RoboDK station: 250418.관통프로젝트준비파일.rdk

Station 250418.관통프로젝트준비파일 (saved by RoboDK 5.9.0). Poses are relative to the parent item; angles as X-Y-Z fixed-axis rotations.
  - Python program RESET (listed below)
  - Python program ADD_File (listed below)
  - notes Note 1: <!DOCTYPE HTML PUBLIC "-//W3C//DTD HTML 4.0//EN" "http://www.w3.org/TR/REC-html40/strict.dtd">
<html><head><meta name="qrichtext" content="1" /><style type="text/css">
p, li { white-space: pre-wrap; }
</style></head><body style=" font-family:'Gulim'; font-size:9pt; font-weight:400; font-style:normal;">
<p style=" margin-top:0px; margin-bottom:0px; margin-left:0px; margin-right:0px; -qt-block-indent:0; text-indent:0px;">관통프로젝트\모델링파일2을 모두 가져옵니다.</p>
<p style=" margin-top:0px; margin-bottom:0px; margin-left:0px; margin-right:0px; -qt-block-indent:0; text-indent:0px;">ADD_File을실행합니다.</p>
<p style=" margin-top:0px; margin-bottom:0px; margin-left:0px; margin-right:0px; -qt-block-indent:0; text-indent:0px;">RESET을 실행합니다.</p></body></html>

--- Python program RESET ---
from robodk import robolink    # RoboDK API
from robodk import robomath    # Robot toolbox
RDK = robolink.Robolink()
from robodk import *      # RoboDK API
from robolink import *    # Robot toolbox










Main_Frame=RDK.Item("Main_Frame",3)
Rack1_Frame=RDK.Item("Rack1 Base",3)
Rack2_Frame=RDK.Item("Rack2 Base",3)
Rack3_Frame=RDK.Item("Rack3 Base",3)
Rack4_Frame=RDK.Item("Rack4 Base",3)

Rack1=RDK.Item("Rack1",2)
Rack2=RDK.Item("Rack2",2)
Rack3=RDK.Item("Rack3",2)
Rack4=RDK.Item("Rack4",2)


Room=RDK.Item("Room",5)

def reset1(): #Room, Rack 위치 설정
      p1=[[     1.000000,     0.000000,     0.000000,     0.000000 ],
            [0.000000,     1.000000,     0.000000,     0.000000 ],
            [0.000000,     0.000000,     1.000000,     0.000000 ],
            [0.000000,     0.000000,     0.000000,     1.000000 ]]
      Room.setParent(Main_Frame)
      Room.setPose(Mat(p1))

      r1=[[     0.000000,     1.000000,     0.000000, -5000.000000 ],
      [-1.000000,     0.000000,     0.000000,  1000.000000 ],
            [0.000000,     0.000000,     1.000000,    50.000000 ],
            [0.000000,     0.000000,     0.000000,     1.000000 ]]


      Rack1_Frame.setPose(Mat(r1))
      Rack2_Frame.setPose(Mat(r1))
      Rack3_Frame.setPose(Mat(r1))
      Rack4_Frame.setPose(Mat(r1))

      Rack1_Frame.setParent(Main_Frame)
      Rack2_Frame.setParent(Main_Frame)
      Rack3_Frame.setParent(Main_Frame)
      Rack4_Frame.setParent(Main_Frame)


      Rack1.setParent(Rack1_Frame)
      Rack2.setParent(Rack2_Frame)
      Rack3.setParent(Rack3_Frame)
      Rack4.setParent(Rack4_Frame)



#####################################


CON1=RDK.Item("CON1",2)
CON1_Frame=RDK.Item("CON1 Base",3)
CON2=RDK.Item("CON2",2)
CON2_Frame=RDK.Item("CON2 Base",3)




def reset2(): #conveyor 위치 설정

      con_pos1=[[     1.000000,     0.000000,     0.000000,   450.000000 ],
      [0.000000,     1.000000,     0.000000,  4000.000000 ],
      [0.000000,     0.000000,     1.000000,   500.000000 ],
      [0.000000,     0.000000,     0.000000,     1.000000 ]]
      con_pos2=[[    -1.000000,     0.000000,     0.000000,   530.000000 ],
     [-0.000000,    -1.000000,     0.000000,  4850.000000 ],
      [0.000000,     0.000000,     1.000000,   500.000000 ],
      [0.000000,     0.000000,     0.000000,     1.000000 ]]

      CON1_Frame.setPose(Mat(con_pos1))
      CON1_Frame.setParent(Main_Frame)
      CON1.setParent(CON1_Frame)

      CON2_Frame.setPose(Mat(con_pos2))
      CON2_Frame.setParent(Main_Frame)
      CON2.setParent(CON2_Frame)

reset1()
reset2()

ABB1_Frame=RDK.Item("ABB1 Base",3)
ABB1_Tool_Frame=RDK.Item("ABB1_Tool Base",3)
ABB1=RDK.Item("ABB1",2)
ABB1_Tool=RDK.Item("ABB1_Tool",4)
ABB1_Base=RDK.Item("ABB1_Setup",5)

p1=[[    -0.642788,    -0.766044,     0.000000, -1750.930000 ],
      [0.766044,    -0.642788,     0.000000,  3081.449000 ],
      [0.000000,     0.000000,     1.000000,   640.000000 ],
      [0.000000,     0.000000,     0.000000,     1.000000 ]]
ABB1_Frame.setParent(Main_Frame)
ABB1_Frame.setPose(Mat(p1))

p2=[[     1.000000,     0.000000,     0.000000,   -69.999988 ],
      [0.000000,     1.000000,     0.000000,    19.999996 ],
      [0.000000,     0.000000,     1.000000,  -590.000000 ],
      [0.000000,     0.000000,     0.000000,     1.000000 ]]



ABB1_Base.setParent(ABB1_Frame)
ABB1_Base.setPose(Mat(p2))

p3=[[     1.000000,    -0.000000,    -0.000000,    -0.000000 ],
     [-0.000000,     0.342020,     0.939693,   194.999972 ],
      [0.000000,    -0.939692,     0.342020,   424.999922 ],
      [0.000000,     0.000000,     0.000000,     1.000000 ]]

ABB1_Tool_Frame.setParent(ABB1)
ABB1_Tool_Frame.setPose(Mat(p3))

--- Python program ADD_File ---
# Type help("robodk.robolink") or help("robodk.robomath") for more information
# Press F5 to run the script
# Documentation: https://robodk.com/doc/en/RoboDK-API.html
# Reference:     https://robodk.com/doc/en/PythonAPI/robodk.html
# Note: It is not required to keep a copy of this file, your Python script is saved with your RDK project

# You can also use the new version of the API:
from robodk import robolink    # RoboDK API
from robodk import robomath    # Robot toolbox
RDK = robolink.Robolink()

# Forward and backwards compatible use of the RoboDK API:
# Remove these 2 lines to follow python programming guidelines
from robodk import *      # RoboDK API
from robolink import *    # Robot toolbox

zero=[[     1.000000,     0.000000,     0.000000,     0.000000 ],
      [0.000000,     1.000000,     0.000000,     0.000000 ],
      [0.000000,     0.000000,     1.000000,     0.000000 ],
      [0.000000,     0.000000,     0.000000,     1.000000 ]]

RDK.AddFrame("Main_Frame")
RDK.AddFrame("Rack1_Work")
RDK.AddFrame("Rack2_Work")
RDK.AddFrame("Rack3_Work")
RDK.AddFrame("Rack4_Work")
RDK.AddFrame("CON1_Work")
RDK.AddFrame("CON2_Work")

RDK.Command("AddFolder", "Rack")
RDK.Command("AddFolder", "Conveyor")

CON1_Work=RDK.Item("CON1_Work",3)
CON2_Work=RDK.Item("CON2_Work",3)

Rack1_Work=RDK.Item("Rack1_Work",3)
Rack2_Work=RDK.Item("Rack2_Work",3)
Rack3_Work=RDK.Item("Rack3_Work",3)
Rack4_Work=RDK.Item("Rack4_Work",3)

Main_Frame=RDK.Item("Main_Frame",3)

Rack1=RDK.Item("Rack1",2)
Rack2=RDK.Item("Rack2",2)
Rack3=RDK.Item("Rack3",2)
Rack4=RDK.Item("Rack4",2)

CON1=RDK.Item("CON1",2)
CON2=RDK.Item("CON2",2)

Main_Frame.setPose(Mat(zero))
CON1_Work.setPose(Mat(zero))
CON2_Work.setPose(Mat(zero))
Rack1_Work.setPose(Mat(zero))
Rack2_Work.setPose(Mat(zero))
Rack3_Work.setPose(Mat(zero))
Rack4_Work.setPose(Mat(zero))

Rack1_Work.setParent(Rack1)
Rack2_Work.setParent(Rack2)
Rack3_Work.setParent(Rack3)
Rack4_Work.setParent(Rack4)

CON1_Work.setParent(CON1)
CON2_Work.setParent(CON2)
